FUNCTION_BLOCK FB_TestSplit EXTENDS TcUnit.FB_TestSuite

testSplit();

METHOD testSplit : BOOL
VAR
	sToSplit		: STRING(255) := 'Hello,this,is,split,test';
	sSplit			: ARRAY[0..Parameters.iSplitArraySize] OF STRING(255);
	sExpected		: ARRAY[0..Parameters.iSplitArraySize] OF STRING(255) := ['Hello', 'this', 'is', 'split', 'test'] ;
	
	i				: INT;
END_VAR
Test('testSplit');
// Arrange

// Act
sSplit := F_STRINGSPLIT(sToSplit, ',');

// Assert
FOR i := 0 TO Parameters.iSplitArraySize DO
	AssertEquals_STRING( Expected := sExpected[i],
				  Actual := sSplit[i],
				  Message := CONCAT('testSplit Failed to split : ', sToSplit));
END_FOR
			 
			 
TEST_FINISHED();
END_METHOD

END_FUNCTION_BLOCK

(* stored: Version 1.1.0.1, ProductVersion 3.1.4024.9
   POU FB_TestSplit: Id {990e2a8f-1f06-451f-ab3b-2f68a8ac23f0}, SpecialFunc None
   Method testSplit: Id {0df167e9-f038-40f0-ac1c-72de488f7c2e} *)
